PROGRAM P_Demo_FB_JsonReadWriteDataType_GetJsonStringFromSymbolProperties
VAR
    fbParser : FB_JsonReadWriteDataType; // 父 FB 实例
    sDatatype : STRING(255);
    sProperties : STRING(255);
    hrErrorCode : HRESULT;
    vRet : STRING(255); // 返回值监视
    bTrigger : BOOL := FALSE; // 在线置 TRUE 触发一次调用
    bTriggerPrev : BOOL;
END_VAR

// =============================================================================
// 场景：从已解析的 JSON DOM 中读取某字段的 JsonStringFromSymbolProperties 类型值（如解析云端下发指令里的目标速度、批次号、状态码）。
// 价值：按节点直接取值，比反复扫字符串快。
// 验证：登录 PLC 在线写 bTrigger := TRUE 触发，monitor 返回值/输出参数。具体步骤见下方注释。
// 验证步骤：
//   1. 右键 PLC 项目下 POUs 文件夹 → Add → Existing Item → 选本 .TcPOU 文件
//   2. 引用 Tc3_JsonXml（References → Add library）
//   3. 编译 → 登录 → 运行；按 verify 注释里给出的在线写值操作
// =============================================================================

// 上升沿触发一次方法调用并观察输出。
IF bTrigger AND NOT bTriggerPrev THEN
    vRet := fbParser.GetJsonStringFromSymbolProperties(
        sDatatype := sDatatype,
        sProperties := sProperties,
        hrErrorCode => hrErrorCode
    );
END_IF;
bTriggerPrev := bTrigger;

END_PROGRAM

(* stored: Version 1.1.0.1, ProductVersion 3.1.4024.5
   POU P_Demo_FB_JsonReadWriteDataType_GetJsonStringFromSymbolProperties: Id {3c2aa79a-fe4b-545b-8ace-8a0ad21cf2da}, SpecialFunc None *)
